// TIA Portal V17 export
// export: Created 2024-06-24T13:40:53.9053686Z, ExportSetting WithDefaults, DisplayName Totally Integrated Automation Portal, DisplayVersion V17, DisplayName TIA Portal Openness, DisplayVersion V17, DisplayName TIA Portal Version Control Interface, DisplayVersion V17, DisplayName STEP 7 Professional, DisplayVersion V17, DisplayName STEP 7 Safety, DisplayVersion V17, DisplayName WinCC Advanced, DisplayVersion V17
VAR_GLOBAL   // PLC tag table "Default tag table"
   alwaysTrue AT %M0.0 : Bool;
   alwaysFalse AT %M1.0 : Bool;
   Tag_1 AT %MW10 : Int;
END_VAR
